TYPE ST_WeighingStation_InOuts :
STRUCT
	stWeighingActuator: ST_ActuatorInOut_TC;
	stPusherActuator: ST_ActuatorInOut_TC;
END_STRUCT
END_TYPE

(* stored: Version 1.1.0.1, ProductVersion 3.1.4024.15
   DUT ST_WeighingStation_InOuts: Id {bb0d82bd-f29e-44e7-8d08-6036991f2cff} *)
